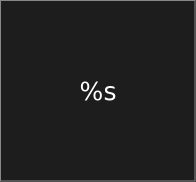
VISUALIZATION Kachel_UWP_Verd  // 196x182
    Rectangle (0,0 196x182), "%s", text list: 'Sprachen', text index: 5
END_VISUALIZATION

// ZY_Visu/Sollwertmenu_9/Wärmegewinnung/Sollwertmenu_Waermegewinnung
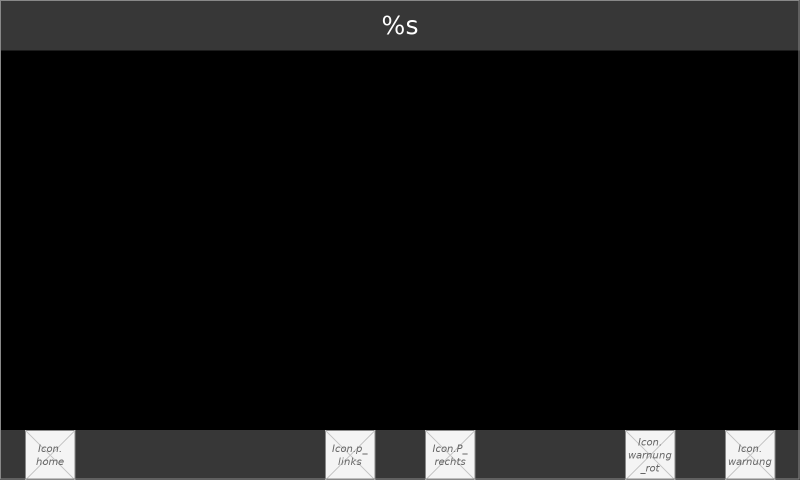
VISUALIZATION Sollwertmenu_Waermegewinnung  // 800x480
VAR_IN_OUT
		
END_VAR

VAR
	i_verschieben:INT;

END_VAR
    Image (425,430 50x50), image: Icon.reinnavigieren
    Image (325,430 50x50), image: Icon.reinnavigieren
    Rectangle (0,0 800x50), "%s", text list: 'Sprachen', text index: 4
    Frame (0,430 800x50)
        shows Fusszeile_50()
    Image (425,430 50x50), image: Icon.P_rechts
        OnMouseClick: execute {
            IF i_verschieben>-800 THEN
            	i_verschieben:=i_verschieben-800;
            END_IF
        }
    Image (325,430 50x50), image: Icon.p_links
        OnMouseClick: execute {
            IF i_verschieben<0 THEN
            	i_verschieben:=i_verschieben+800;
            END_IF
        }
    Rectangle (88,515 454x57), "Kachel 1: 0;55 *** Kachel 2: 201;55 *** Kachel 3: 402;55 *** Kachel 4: 604;55 Kachel 5: 0;242 *** Kachel 6: 201;242 *** Kachel 7: 402;242 *** Kachel 8: 604;242"
END_VISUALIZATION

// ZY_Visu/Sollwertmenu_9/Wärmepumpe/EEV/SW_WP_EEV
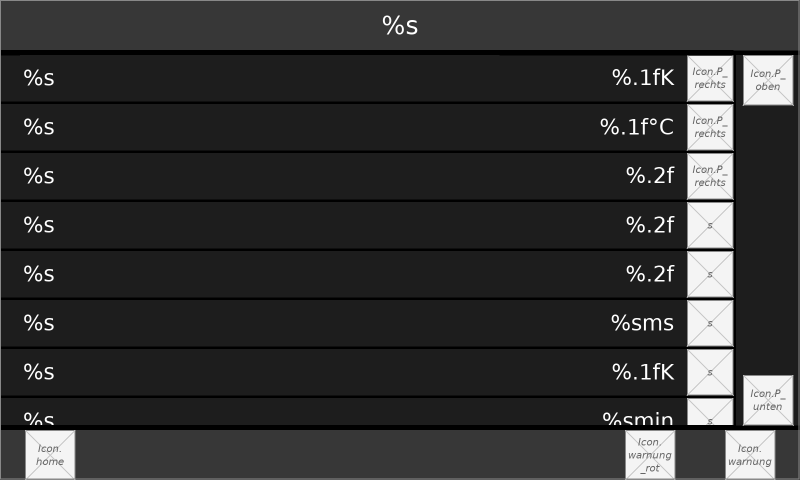
VISUALIZATION SW_WP_EEV  // 800x480
VAR_IN_OUT
	FB_EEV:EEV;
	
END_VAR
	
VAR_INPUT
	

END_VAR
    Frame (0,0 800x430), frame switch variable: GWP_Library.Visu.i_Frame_Index
        shows SW_WP_EEV_Liste(i_Titel := 15, FB_EEV := FB_EEV)
        shows SW_Einstellungen_K(i_titel := 30, f_Data := FB_EEV.f_SollwertUBH)
        shows SW_Einstellungen_C(i_titel := 30, f_Data := FB_EEV.f_MOP)
        shows SW_Einstellungen_Faktor(i_titel := 30, f_Data := FB_EEV.f_PFaktor)
        shows SW_Einstellungen_Faktor(i_titel := 30, f_Data := FB_EEV.f_IFaktor)
        shows SW_Einstellungen_Faktor(i_titel := 30, f_Data := FB_EEV.f_DFaktor)
        shows SW_Einstellungen_ms(i_titel := 30, f_Data := FB_EEV.t_Takt.wMilliseconds)
        shows SW_Einstellungen_K(i_titel := 30, f_Data := FB_EEV.f_MinUBH)
        shows SW_Einstellungen_min(i_titel := 30, f_Data := FB_EEV.t_AL_EEV.wMinute)
        shows SW_zuruecksetzen(i_Titel := 72, i_Text_1 := 73, i_Text_2 := 72, x_Zuruecksetzen := FB_EEV.x_SW_Reset)
    Frame (0,430 800x50)
        shows Fusszeile_50()
END_VISUALIZATION

// ZY_Visu/Sollwertmenu_9/Wärmepumpe/EEV/SW_WP_EEV_Liste
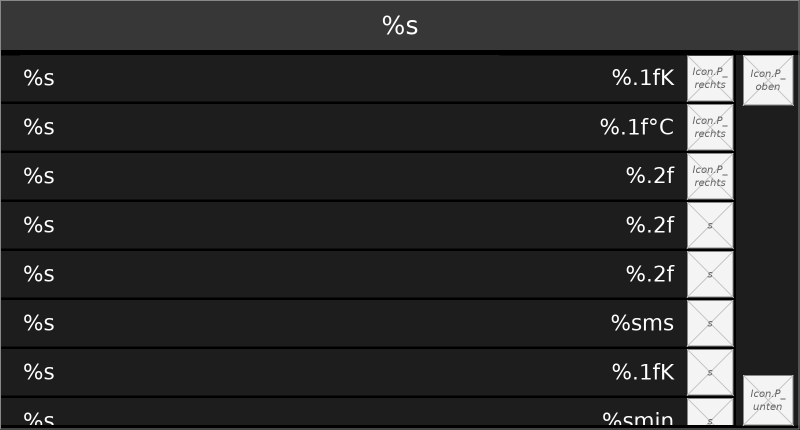
VISUALIZATION SW_WP_EEV_Liste  // 800x430
VAR_IN_OUT
	FB_EEV:EEV;	
	
END_VAR
	
VAR_INPUT
	i_Titel:INT;

END_VAR

VAR
	i_ref_versch:INT;
END_VAR
    Rectangle (0,0 800x50), "%s", text list: 'Sprachen', text index: i_Titel
    Rectangle (736,55 64x370)
    Image (743,375 50x50), image: Icon.P_unten
        OnMouseClick: execute { i_ref_versch:=i_ref_versch + 53; }
    Image (743,55 50x50), image: Icon.P_oben
        OnMouseClick: execute { i_ref_versch:=i_ref_versch - 53; }
    Rectangle (0,55 733x46)
    Rectangle (0,104 733x46)
    Rectangle (547,55 130x45), "%.1fK", text variable: FB_EEV.f_SollwertUBH
    Rectangle (547,104 130x46), "%.1f°C", text variable: FB_EEV.f_MOP
    Image (687,55 46x46), image: Icon.P_rechts
        OnMouseClick: execute { Visu.i_Frame_Index:=1; }
    Image (687,104 46x46), image: Icon.P_rechts
        OnMouseClick: execute { Visu.i_Frame_Index:=2; }
    Rectangle (0,153 733x46)
    Rectangle (0,202 733x46)
    Rectangle (0,251 733x46)
    Rectangle (0,300 733x46)
    Rectangle (0,349 733x46)
    Rectangle (0,398 733x46)
    Rectangle (0,447 733x46)
    Rectangle (0,496 733x46)
    Rectangle (0,545 733x46)
    Rectangle (547,153 130x45), "%.2f", text variable: FB_EEV.f_PFaktor
        OnMouseClick: execute { GWP_Library.Visu.i_Frame_Index:=2; }
    Rectangle (547,202 130x46), "%.2f", text variable: FB_EEV.f_IFaktor
    Rectangle (547,251 130x46), "%.2f", text variable: FB_EEV.f_DFaktor
    Rectangle (547,300 130x46), "%sms", text variable: FB_EEV.t_Takt.wMilliseconds
    Rectangle (547,349 130x46), "%.1fK", text variable: FB_EEV.f_MinUBH
    Rectangle (547,398 130x46), "%smin", text variable: FB_EEV.t_AL_EEV.wMinute
    Rectangle (547,496 130x46), "Ein"
    Rectangle (547,545 130x46), "Ein"
    Image (687,153 46x46), image: Icon.P_rechts
        OnMouseClick: execute { GWP_Library.Visu.i_Frame_Index:=3; }
    Image (687,545 46x46), image: s
    Image (687,496 46x46), image: Icon.P_rechts
    Image (687,447 46x46), image: Icon.P_rechts
        OnMouseClick: execute { GWP_Library.Visu.i_Frame_Index:=9; }
    Image (687,398 46x46), image: s
        OnMouseClick: execute { GWP_Library.Visu.i_Frame_Index:=8; }
    Image (687,349 46x46), image: s
        OnMouseClick: execute { GWP_Library.Visu.i_Frame_Index:=7; }
    Image (687,300 46x46), image: s
        OnMouseClick: execute { GWP_Library.Visu.i_Frame_Index:=6; }
    Image (687,251 46x46), image: s
        OnMouseClick: execute { GWP_Library.Visu.i_Frame_Index:=5; }
    Image (687,202 46x46), image: s
        OnMouseClick: execute { GWP_Library.Visu.i_Frame_Index:=4; }
    Rectangle (0,594 733x46)
    Rectangle (547,594 130x45), "Ein"
    Image (687,594 46x46), image: Icon.P_rechts
    Image (79,430 50x50), image: Icon.zurueck
        OnMouseClick:  Assign=Sollwertmenu_Waermegewinnung, Type=Assignment
        OnMouseClick: execute { i_verschieben:=0; }
    Rectangle (0,50 733x5)
    Rectangle (20,55 479x46), "%s", text list: 'Sprachen', text index: 85
    Rectangle (20,104 479x46), "%s", text list: 'Sprachen', text index: 86
    Rectangle (20,202 479x46), "%s", text list: 'Sprachen', text index: 88
    Rectangle (20,153 479x46), "%s", text list: 'Sprachen', text index: 87
    Rectangle (20,251 479x46), "%s", text list: 'Sprachen', text index: 89
    Rectangle (20,300 479x46), "%s", text list: 'Sprachen', text index: 90
    Rectangle (20,349 479x46), "%s", text list: 'Sprachen', text index: 91
    Rectangle (20,398 479x46), "%s", text list: 'Sprachen', text index: 92
    Rectangle (20,447 479x46), "%s", text list: 'Sprachen', text index: 72
    Rectangle (20,496 479x46), "%s", text list: 'Sprachen'
    Rectangle (20,545 479x46), "%s", text list: 'Sprachen'
    Rectangle (20,594 479x46), "%s", text list: 'Sprachen'
    Rectangle (0,425 733x5)
END_VISUALIZATION

// ZY_Visu/Sollwertmenu_9/Wärmepumpe/Einsatzgrenzen/SW_WP_Einsatzgrenzen
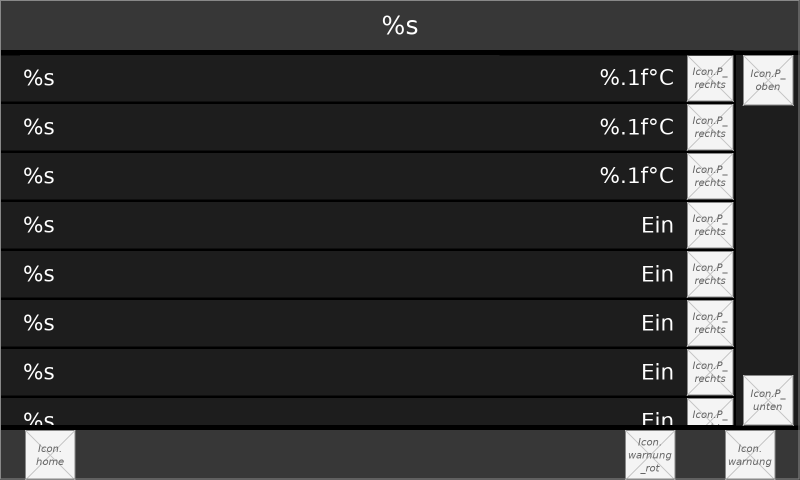
VISUALIZATION SW_WP_Einsatzgrenzen  // 800x480
VAR_IN_OUT
	FB_Einsatzgrenzen:Einsatzgrenzen;
END_VAR
    Frame (0,0 800x430)
        shows SW_WP_Einsatzgrenzen_Liste(i_Titel := 21, FB_Einsatzgrenzen := FB_Einsatzgrenzen)
    Frame (0,430 800x50)
        shows Fusszeile_50()
END_VISUALIZATION

// ZY_Visu/Sollwertmenu_9/Wärmepumpe/Einsatzgrenzen/SW_WP_Einsatzgrenzen_Liste
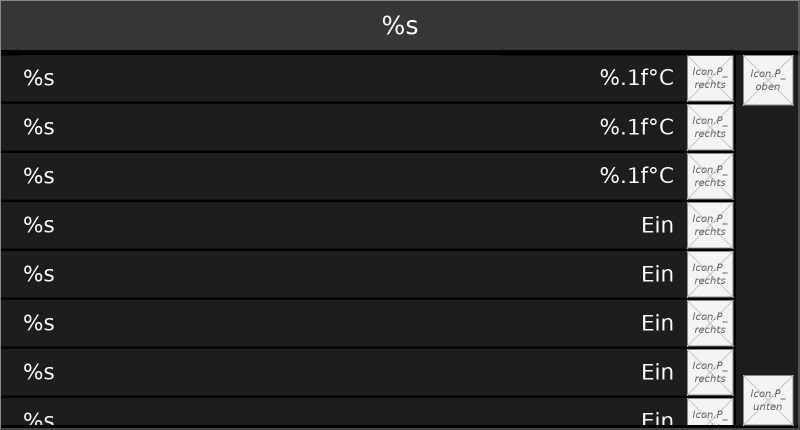
VISUALIZATION SW_WP_Einsatzgrenzen_Liste  // 800x430
VAR_IN_OUT
	FB_Einsatzgrenzen:Einsatzgrenzen;
END_VAR

VAR_INPUT
	i_Titel:INT;
END_VAR

VAR
	i_verschieben:INT;
 END_VAR
    Rectangle (0,55 733x46)
    Rectangle (0,104 733x46)
    Rectangle (547,55 130x45), "%.1f°C", text variable: FB_EEV.f_Regelsignal
    Rectangle (547,104 130x46), "%.1f°C"
    Image (687,55 46x46), image: Icon.P_rechts
        OnMouseClick: execute { Visu.i_Frame_Index:=1; }
    Image (687,104 46x46), image: Icon.P_rechts
        OnMouseClick: execute { Visu.i_Frame_Index:=2; }
    Rectangle (0,153 733x46)
    Rectangle (0,202 733x46)
    Rectangle (0,251 733x46)
    Rectangle (0,300 733x46)
    Rectangle (0,349 733x46)
    Rectangle (0,398 733x46)
    Rectangle (0,447 733x46)
    Rectangle (0,496 733x46)
    Rectangle (0,545 733x46)
    Rectangle (547,153 130x45), "%.1f°C"
        OnMouseClick: execute { GWP_Library.Visu.i_Frame_Index:=2; }
    Rectangle (547,202 130x46), "Ein"
    Rectangle (547,251 130x46), "Ein"
    Rectangle (547,300 130x46), "Ein"
    Rectangle (547,349 130x46), "Ein"
    Rectangle (547,447 130x46), "Ein"
    Rectangle (547,398 130x46), "Ein"
    Rectangle (547,496 130x46), "Ein"
    Rectangle (547,545 130x46), "Ein"
    Image (687,153 46x46), image: Icon.P_rechts
        OnMouseClick: execute { GWP_Library.Visu.i_Frame_Index:=3; }
    Image (687,545 46x46), image: s
    Image (687,496 46x46), image: Icon.P_rechts
    Image (687,447 46x46), image: Icon.P_rechts
    Image (687,398 46x46), image: Icon.P_rechts
    Image (687,349 46x46), image: Icon.P_rechts
    Image (687,300 46x46), image: Icon.P_rechts
    Image (687,251 46x46), image: Icon.P_rechts
    Image (687,202 46x46), image: Icon.P_rechts
    Rectangle (0,594 733x46)
    Rectangle (547,594 130x45), "Ein"
    Image (687,594 46x46), image: Icon.P_rechts
    Image (79,430 50x50), image: Icon.zurueck
        OnMouseClick:  Assign=Sollwertmenu_Waermegewinnung, Type=Assignment
        OnMouseClick: execute { i_verschieben:=0; }
    Rectangle (0,0 800x50), "%s", text list: 'Sprachen', text index: i_Titel
    Rectangle (736,55 64x370)
    Image (743,375 50x50), image: Icon.P_unten
        OnMouseClick: execute {
            IF i_verschieben<0 THEN
            	i_verschieben:=i_verschieben+53;
            End_if
        }
    Image (743,55 50x50), image: Icon.P_oben
        OnMouseClick: execute {
            IF  i_verschieben>-200 THEN
            	i_verschieben:=i_verschieben-53;
            End_if
        }
    Rectangle (0,50 733x5)
    Rectangle (20,55 479x46), "%s", text list: 'Sprachen'
    Rectangle (20,104 479x46), "%s", text list: 'Sprachen'
    Rectangle (20,202 479x46), "%s", text list: 'Sprachen'
    Rectangle (20,153 479x46), "%s", text list: 'Sprachen'
    Rectangle (20,251 479x46), "%s", text list: 'Sprachen'
    Rectangle (20,300 479x46), "%s", text list: 'Sprachen'
    Rectangle (20,349 479x46), "%s", text list: 'Sprachen'
    Rectangle (20,398 479x46), "%s", text list: 'Sprachen'
    Rectangle (20,447 479x46), "%s", text list: 'Sprachen'
    Rectangle (20,496 479x46), "%s", text list: 'Sprachen'
    Rectangle (20,545 479x46), "%s", text list: 'Sprachen'
    Rectangle (20,594 479x46), "%s", text list: 'Sprachen'
    Rectangle (0,425 733x5)
END_VISUALIZATION

// ZY_Visu/Sollwertmenu_9/Wärmepumpe/Kachel_Allgemein
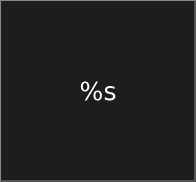
VISUALIZATION Kachel_Allgemein  // 196x182
    Rectangle (0,0 196x182), "%s", text list: 'Sprachen', text index: 18
END_VISUALIZATION

// ZY_Visu/Sollwertmenu_9/Wärmepumpe/Kachel_EEV
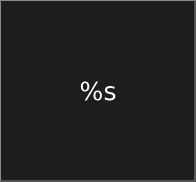
VISUALIZATION Kachel_EEV  // 196x182
    Rectangle (0,0 196x182), "%s", text list: 'Sprachen', text index: 15
END_VISUALIZATION

// ZY_Visu/Sollwertmenu_9/Wärmepumpe/Kachel_Einsatzgrenzen
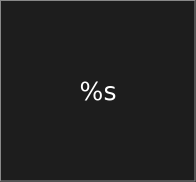
VISUALIZATION Kachel_Einsatzgrenzen  // 196x182
    Rectangle (0,0 196x182), "%s", text list: 'Sprachen', text index: 16
END_VISUALIZATION

// ZY_Visu/Sollwertmenu_9/Wärmepumpe/Kachel_Verdichter
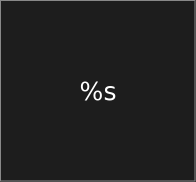
VISUALIZATION Kachel_Verdichter  // 196x182
    Rectangle (0,0 196x182), "%s", text list: 'Sprachen', text index: 17
END_VISUALIZATION

// ZY_Visu/Sollwertmenu_9/Wärmepumpe/Sollwertmenu_Waermepumpe
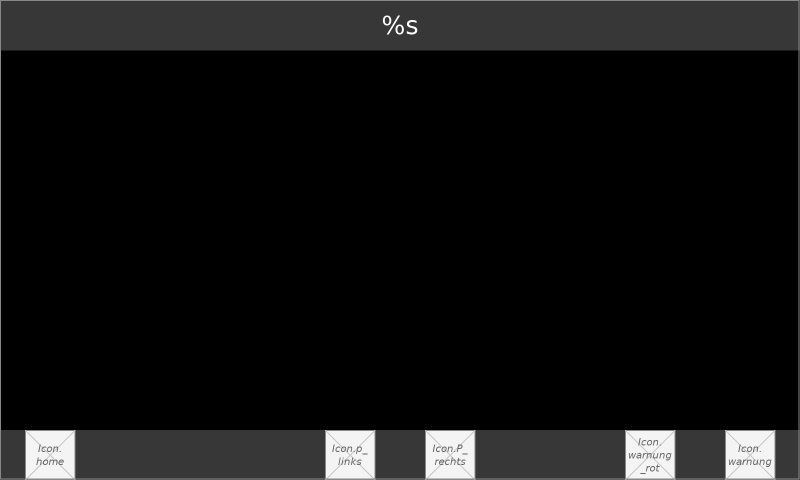
VISUALIZATION Sollwertmenu_Waermepumpe  // 800x480
VAR_IN_OUT
		
END_VAR

VAR
	i_verschieben:INT;

END_VAR
    Image (425,430 50x50), image: Icon.reinnavigieren
    Image (325,430 50x50), image: Icon.reinnavigieren
    Rectangle (0,0 800x50), "%s", text list: 'Sprachen', text index: 14
    Frame (0,430 800x50)
        shows Fusszeile_50()
    Image (425,430 50x50), image: Icon.P_rechts
        OnMouseClick: execute {
            IF i_verschieben>-800 THEN
            	i_verschieben:=i_verschieben-800;
            END_IF
        }
    Image (325,430 50x50), image: Icon.p_links
        OnMouseClick: execute {
            IF i_verschieben<0 THEN
            	i_verschieben:=i_verschieben+800;
            END_IF
        }
    Rectangle (88,515 454x57), "Kachel 1: 0;55 *** Kachel 2: 201;55 *** Kachel 3: 402;55 *** Kachel 4: 604;55 Kachel 5: 0;242 *** Kachel 6: 201;242 *** Kachel 7: 402;242 *** Kachel 8: 604;242"
END_VISUALIZATION

// ZY_Visu/Sollwertmenu_9/Wärmesenke/Kachel_Heizgruppen
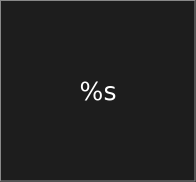
VISUALIZATION Kachel_Heizgruppen  // 196x182
    Rectangle (0,0 196x182), "%s", text list: 'Sprachen', text index: 23
END_VISUALIZATION

// ZY_Visu/Sollwertmenu_9/Wärmesenke/Kachel_Hochhaltung
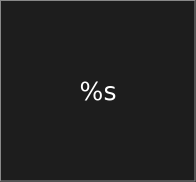
VISUALIZATION Kachel_Hochhaltung  // 196x182
    Rectangle (0,0 196x182), "%s", text list: 'Sprachen', text index: 24
END_VISUALIZATION

// ZY_Visu/Sollwertmenu_9/Wärmesenke/Kachel_HWP
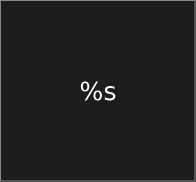
VISUALIZATION Kachel_HWP  // 196x182
    Rectangle (0,0 196x182), "%s", text list: 'Sprachen', text index: 21
END_VISUALIZATION

// ZY_Visu/Sollwertmenu_9/Wärmesenke/Kachel_TWW
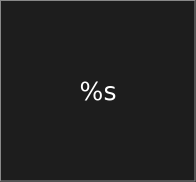
VISUALIZATION Kachel_TWW  // 196x182
    Rectangle (0,0 196x182), "%s", text list: 'Sprachen', text index: 22
END_VISUALIZATION

// ZY_Visu/Sollwertmenu_9/Wärmesenke/Kachel_UWP_Verfl
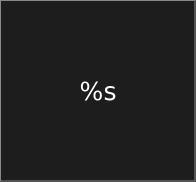
VISUALIZATION Kachel_UWP_Verfl  // 196x182
    Rectangle (0,0 196x182), "%s", text list: 'Sprachen', text index: 20
END_VISUALIZATION

// ZY_Visu/Sollwertmenu_9/Wärmesenke/Sollwertmenu_Waermesenke
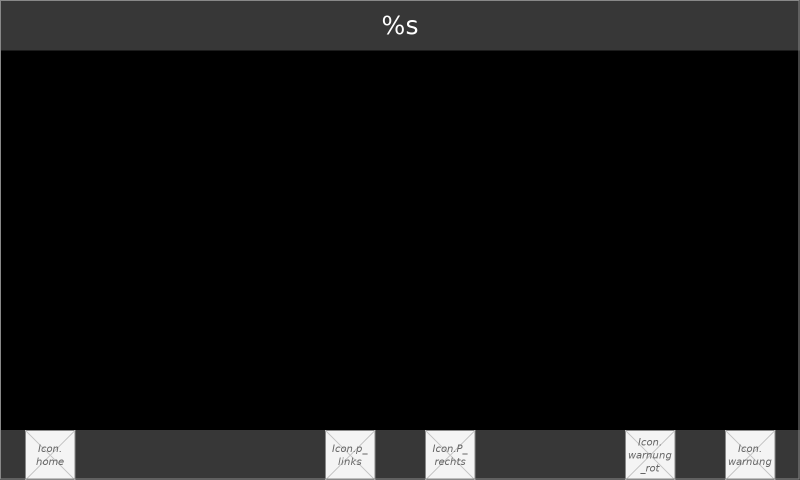
VISUALIZATION Sollwertmenu_Waermesenke  // 800x480
VAR_IN_OUT
		
END_VAR

VAR
	i_verschieben:INT;

END_VAR
    Image (425,430 50x50), image: Icon.reinnavigieren
    Image (325,430 50x50), image: Icon.reinnavigieren
    Rectangle (0,0 800x50), "%s", text list: 'Sprachen', text index: 19
    Frame (0,430 800x50)
        shows Fusszeile_50()
    Image (425,430 50x50), image: Icon.P_rechts
        OnMouseClick: execute {
            IF i_verschieben>-800 THEN
            	i_verschieben:=i_verschieben-800;
            END_IF
        }
    Image (325,430 50x50), image: Icon.p_links
        OnMouseClick: execute {
            IF i_verschieben<0 THEN
            	i_verschieben:=i_verschieben+800;
            END_IF
        }
    Rectangle (88,515 483x57), "Kachel 1: 0;55 *** Kachel 2: 201;55 *** Kachel 3: 402;55 *** Kachel 4: 604;55 Kachel 5: 0;242 *** Kachel 6: 201;242 *** Kachel 7: 402;242 *** Kachel 8: 604;242"
END_VISUALIZATION

// ZY_Visu/Sprache/Spracheistellungen
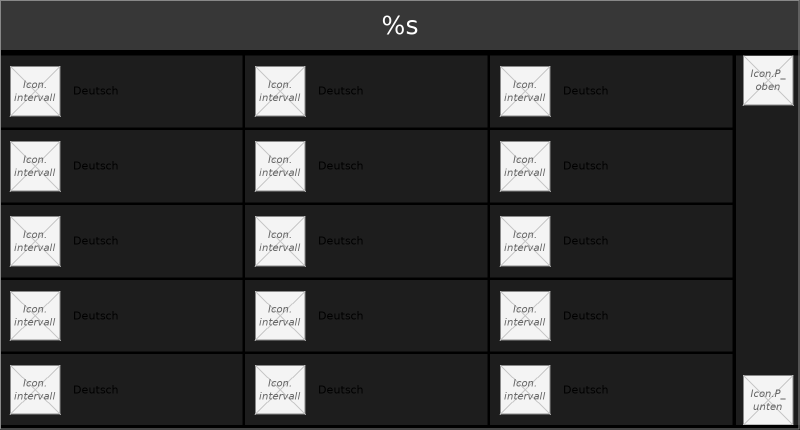
VISUALIZATION Spracheistellungen  // 800x430
VAR_IN_OUT

END_VAR

VAR_INPUT
	
END_VAR

VAR
	i_verschieben:INT;
 END_VAR
    Group (0,55 732x743)
        p2738717112: i_verschieben
        Rectangle (490,0 242x72)
        Rectangle (560,18 151x36), "Deutsch"
        Image (500,11 50x50), image: Icon.intervall
        Rectangle (245,0 242x72)
        Rectangle (315,18 151x36), "Deutsch"
        Image (255,11 50x50), image: Icon.intervall
        Rectangle (0,0 242x72)
        Rectangle (70,18 151x36), "Deutsch"
        Image (10,11 50x50), image: Icon.intervall
        Rectangle (490,75 242x72)
        Rectangle (560,93 151x36), "Deutsch"
        Image (500,86 50x50), image: Icon.intervall
        Rectangle (245,75 242x72)
        Rectangle (315,93 151x36), "Deutsch"
        Image (255,86 50x50), image: Icon.intervall
        Rectangle (0,75 242x72)
        Rectangle (70,93 151x36), "Deutsch"
        Image (10,86 50x50), image: Icon.intervall
        Rectangle (490,150 242x72)
        Rectangle (560,168 151x36), "Deutsch"
        Image (500,161 50x50), image: Icon.intervall
        Rectangle (245,150 242x72)
        Rectangle (315,168 151x36), "Deutsch"
        Image (255,161 50x50), image: Icon.intervall
        Rectangle (0,150 242x72)
        Rectangle (70,168 151x36), "Deutsch"
        Image (10,161 50x50), image: Icon.intervall
        Rectangle (490,225 242x71)
        Rectangle (560,243 151x36), "Deutsch"
        Image (500,236 50x49), image: Icon.intervall
        Rectangle (245,225 242x71)
        Rectangle (315,243 151x36), "Deutsch"
        Image (255,236 50x49), image: Icon.intervall
        Rectangle (0,225 242x71)
        Rectangle (70,243 151x36), "Deutsch"
        Image (10,236 50x49), image: Icon.intervall
        Rectangle (490,299 242x71)
        Rectangle (560,317 151x36), "Deutsch"
        Image (500,310 50x49), image: Icon.intervall
        Rectangle (245,299 242x71)
        Rectangle (315,317 151x36), "Deutsch"
        Image (255,310 50x49), image: Icon.intervall
        Rectangle (0,299 242x71)
        Rectangle (70,317 151x36), "Deutsch"
        Image (10,310 50x49), image: Icon.intervall
        Rectangle (490,373 242x72)
        Rectangle (560,391 151x36), "Deutsch"
        Image (500,384 50x50), image: Icon.intervall
        Rectangle (245,373 242x72)
        Rectangle (315,391 151x36), "Deutsch"
        Image (255,384 50x50), image: Icon.intervall
        Rectangle (0,373 242x72)
        Rectangle (70,391 151x36), "Deutsch"
        Image (10,384 50x50), image: Icon.intervall
        Rectangle (490,448 242x72)
        Rectangle (560,466 151x36), "Deutsch"
        Image (500,459 50x50), image: Icon.intervall
        Rectangle (245,448 242x72)
        Rectangle (315,466 151x36), "Deutsch"
        Image (255,459 50x50), image: Icon.intervall
        Rectangle (0,448 242x72)
        Rectangle (70,466 151x36), "Deutsch"
        Image (10,459 50x50), image: Icon.intervall
        Rectangle (490,523 242x72)
        Rectangle (560,541 151x36), "Deutsch"
        Image (500,534 50x50), image: Icon.intervall
        Rectangle (245,523 242x72)
        Rectangle (315,541 151x36), "Deutsch"
        Image (255,534 50x50), image: Icon.intervall
        Rectangle (0,523 242x72)
        Rectangle (70,541 151x36), "Deutsch"
        Image (10,534 50x50), image: Icon.intervall
        Rectangle (490,598 242x71)
        Rectangle (560,616 151x36), "Deutsch"
        Image (500,609 50x49), image: Icon.intervall
        Rectangle (245,598 242x71)
        Rectangle (315,616 151x36), "Deutsch"
        Image (255,609 50x49), image: Icon.intervall
        Rectangle (0,598 242x71)
        Rectangle (70,616 151x36), "Deutsch"
        Image (10,609 50x49), image: Icon.intervall
        Rectangle (490,672 242x71)
        Rectangle (560,690 151x36), "Deutsch"
        Image (500,683 50x49), image: Icon.intervall
        Rectangle (245,672 242x71)
        Rectangle (315,690 151x36), "Deutsch"
        Image (255,683 50x49), image: Icon.intervall
        Rectangle (0,672 242x71)
        Rectangle (70,690 151x36), "Deutsch"
        Image (10,683 50x49), image: Icon.intervall
    Rectangle (0,0 800x50), "%s", text list: 'Sprachen', text index: 70
    Group (736,55 64x370)
        Rectangle (0,0 64x370)
        Image (7,320 50x50), image: Icon.P_unten
            OnMouseClick: execute {
                IF i_verschieben<0 THEN
                	i_verschieben:=i_verschieben+75;
                End_if
            }
        Image (7,0 50x50), image: Icon.P_oben
            OnMouseClick: execute {
                IF  i_verschieben>-375 THEN
                	i_verschieben:=i_verschieben-75;
                End_if
            }
    Frame (0,430 800x50)
        shows Fusszeile_50()
    Rectangle (0,50 800x5)
    Rectangle (0,425 800x5)
END_VISUALIZATION

// ZY_Visu/Zeitprogramm/Aenderung_Zeit/Ein_Aus_Zeit_aendern
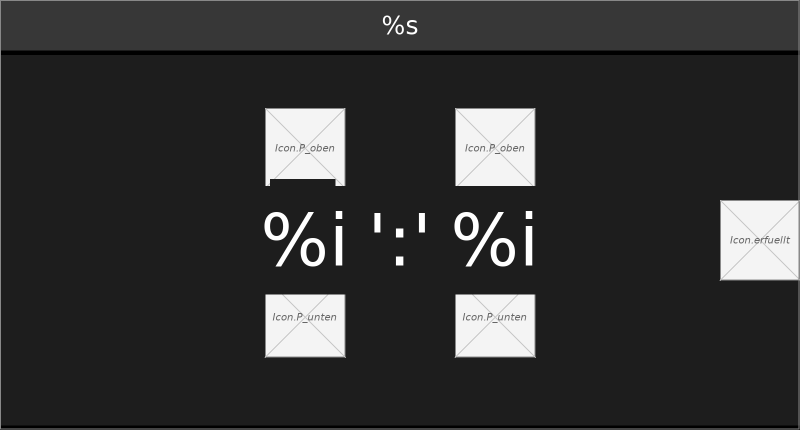
VISUALIZATION Ein_Aus_Zeit_aendern  // 800x430
VAR

END_VAR
VAR_IN_OUT
	i_Minuten:WORD;
	i_Stunden:WORD;	
END_VAR

VAR_INPUT
	i_titel:INT;
END_VAR
    Rectangle (0,0 800x50), "%s", text list: 'Sprachen', text index: i_titel
    Rectangle (0,55 800x370)
    Image (720,200 80x80), image: Icon.erfuellt
        OnMouseClick: execute { Visu.i_Frame_Index:=0; }
    Image (265,108 80x80), image: Icon.P_oben
        OnMouseClick: execute { i_Stunden:=i_Stunden +1; }
    Image (455,108 80x80), image: Icon.P_oben
        OnMouseClick: execute { i_Minuten:=i_Minuten +1; }
    Image (265,277 80x80), image: Icon.P_unten
        OnMouseClick: execute { i_Stunden:=i_Stunden -1; }
    Image (455,277 80x80), image: Icon.P_unten
        OnMouseClick: execute { i_Minuten:=i_Minuten -1; }
    Rectangle (420,186 150x108), "%i", text variable: i_Minuten
    Rectangle (270,179 65x105)
    Rectangle (230,186 150x108), "%i", text variable: i_Stunden
    Rectangle (395,186 10x108), "':'"
END_VISUALIZATION

// ZY_Visu/Zeitprogramm/Aenderung_Zeit/Monat_aendern
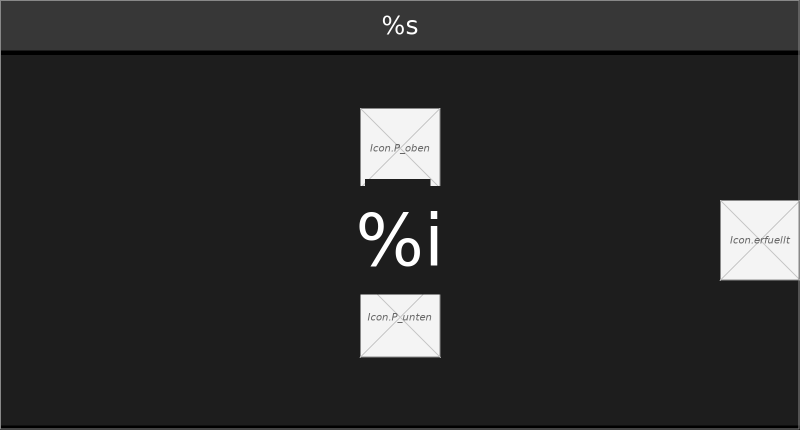
VISUALIZATION Monat_aendern  // 800x430
VAR

END_VAR
VAR_IN_OUT
	i_Monat:WORD;

END_VAR

VAR_INPUT
	i_titel:INT;
END_VAR
    Rectangle (0,0 800x50), "%s", text list: 'Sprachen', text index: i_titel
    Rectangle (0,55 800x370)
    Image (720,200 80x80), image: Icon.erfuellt
        OnMouseClick: execute { Visu.i_Frame_Index:=0; }
    Image (360,108 80x80), image: Icon.P_oben
        OnMouseClick: execute { i_Monat:=i_Monat +1; }
    Image (360,277 80x80), image: Icon.P_unten
        OnMouseClick: execute { i_Monat:=i_Monat -1; }
    Rectangle (365,179 65x105)
    Rectangle (325,186 150x108), "%i", text variable: i_Monat
END_VISUALIZATION

// ZY_Visu/Zeitprogramm/Aenderung_Zeit/Monatstag_aendern
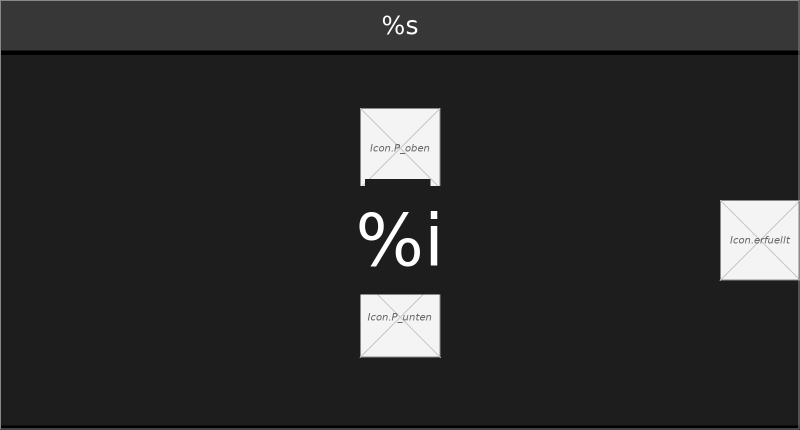
VISUALIZATION Monatstag_aendern  // 800x430
VAR

END_VAR
VAR_IN_OUT
	i_Monatstag:WORD;

END_VAR

VAR_INPUT
	i_titel:INT;
END_VAR
    Rectangle (0,0 800x50), "%s", text list: 'Sprachen', text index: i_titel
    Rectangle (0,55 800x370)
    Image (720,200 80x80), image: Icon.erfuellt
        OnMouseClick: execute { Visu.i_Frame_Index:=0; }
    Image (360,108 80x80), image: Icon.P_oben
        OnMouseClick: execute { i_Monatstag:=i_Monatstag +1; }
    Image (360,277 80x80), image: Icon.P_unten
        OnMouseClick: execute { i_Monatstag:=i_Monatstag -1; }
    Rectangle (365,179 65x105)
    Rectangle (325,186 150x108), "%i", text variable: i_Monatstag
END_VISUALIZATION

// ZY_Visu/Zeitprogramm/Aenderung_Zeit/Sekunden_aendern
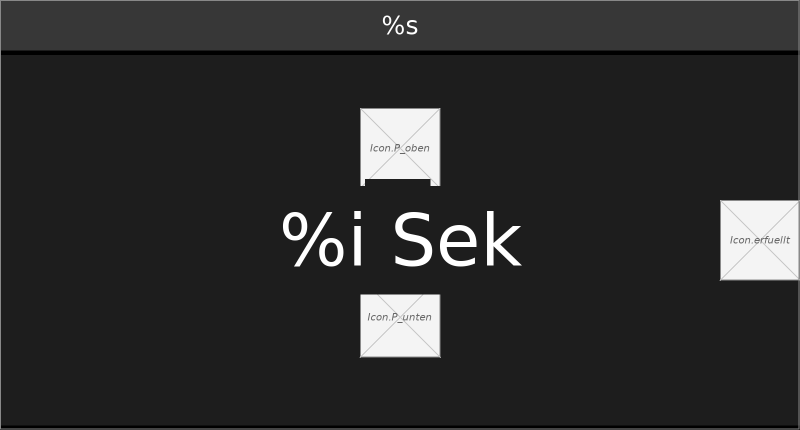
VISUALIZATION Sekunden_aendern  // 800x430
VAR

END_VAR
VAR_IN_OUT
	i_Sekunden:WORD;

END_VAR

VAR_INPUT
	i_titel:INT;
END_VAR
    Rectangle (0,0 800x50), "%s", text list: 'Sprachen', text index: i_titel
    Rectangle (0,55 800x370)
    Image (720,200 80x80), image: Icon.erfuellt
        OnMouseClick: execute { Visu.i_Frame_Index:=0; }
    Image (360,108 80x80), image: Icon.P_oben
        OnMouseClick: execute { i_Sekunden:=i_Sekunden +1; }
    Image (360,277 80x80), image: Icon.P_unten
        OnMouseClick: execute { i_Sekunden:=i_Sekunden -1; }
    Rectangle (365,179 65x105)
    Rectangle (182,186 437x108), "%i Sek", text variable: i_Sekunden
END_VISUALIZATION

// ZY_Visu/Zeitprogramm/Aenderung_Zeit/Wochentag_aendern
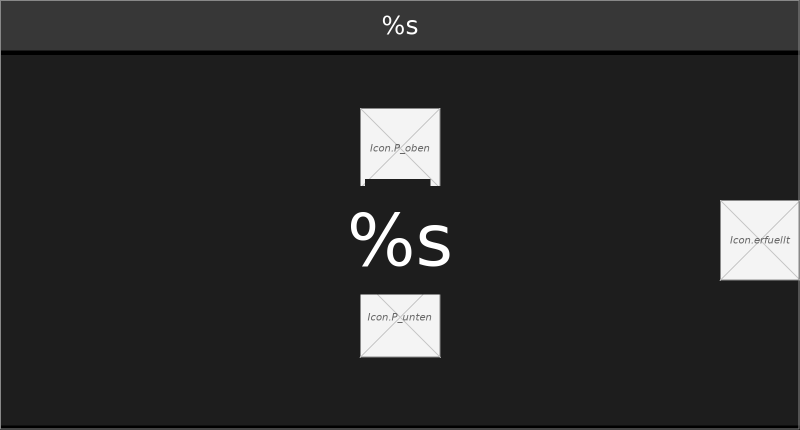
VISUALIZATION Wochentag_aendern  // 800x430
VAR
	
	
END_VAR
VAR_IN_OUT
	i_Wochentag:WORD;

END_VAR

VAR_INPUT
	i_titel:INT;
END_VAR
    Rectangle (0,0 800x50), "%s", text list: 'Sprachen', text index: i_titel
    Rectangle (0,55 800x370)
    Image (720,200 80x80), image: Icon.erfuellt
        OnMouseClick: execute { Visu.i_Frame_Index:=0; }
    Image (360,108 80x80), image: Icon.P_oben
        OnMouseClick: execute { i_Wochentag:=i_Wochentag +1; }
    Image (360,277 80x80), image: Icon.P_unten
        OnMouseClick: execute { i_Wochentag:=i_Wochentag -1; }
    Rectangle (365,179 65x105)
    Rectangle (325,186 150x108), "%s", text variable: i_Wochentag
END_VISUALIZATION

// ZY_Visu/Zeitprogramm/CLK_D/CLK_D_Tagesprogramm
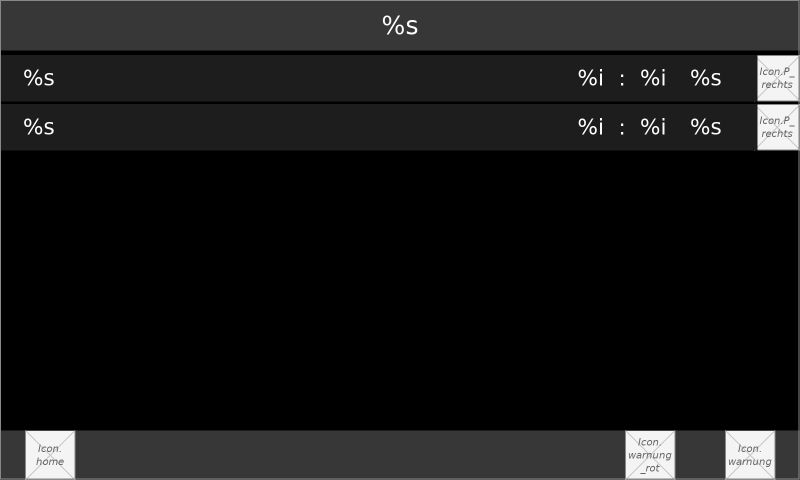
VISUALIZATION CLK_D_Tagesprogramm  // 800x480
VAR_IN_OUT
	FB_CLK_D:CLK_D;

END_VAR
    Frame (0,430 800x50)
        shows Fusszeile_50()
    Frame (0,0 800x430), frame switch variable: Visu.i_Frame_Index
        shows CLK_D_Tagesprogramm_Liste(i_Titel := 77, FB_CLK_D := FB_CLK_D)
        shows Ein_Aus_Zeit_aendern(i_titel := 68, i_Minuten := FB_CLK_D.t_Ein.wMinute, i_Stunden := FB_CLK_D.t_Ein.wHour)
        shows Ein_Aus_Zeit_aendern(i_titel := 68, i_Minuten := FB_CLK_D.t_Aus.wMinute, i_Stunden := FB_CLK_D.t_Aus.wHour)
END_VISUALIZATION

// ZY_Visu/Zeitprogramm/CLK_D/CLK_D_Tagesprogramm_Liste
